(* Schneider Machine Expert - Basic project A7 Temporizador TOF, file version 2.7.0.0 *)
(* ProjectInformations: Name=Novo projeto *)

HARDWARE
  Cpu 0: TM221M16R/G
  EthernetConfiguration: NetworkName=M221, IpAllocationMode=FixedAddress, IpAddress=0.0.0.0, SubnetMask=0.0.0.0
  SerialLineConfiguration: Baud=Baud19200, Parity=ParityEven, DataBits=DataBits8, StopBits=StopBits1, PhysicalMedium=PhysicalMediumRs485, TransmissionMode=TransmissionModeModbusRtu, SlaveId=1, Addressing=SlaveAddressing
  MastTask: UsePeriodScanMode=false, PeriodScan=100
  FastTask: Period=255
  CpuBehavior: StartingMode=StartAsPreviousState, AutoSaveRamOnEeprom=true, WatchdogPeriod=250

SYMBOLS  (address, symbol, comment, settings)
  %TM0        [Type=TOF, Preset=10, Base=OneSecond, IsRetentive=true]

POU Novo POU
  (* SectionNumber=1 *)

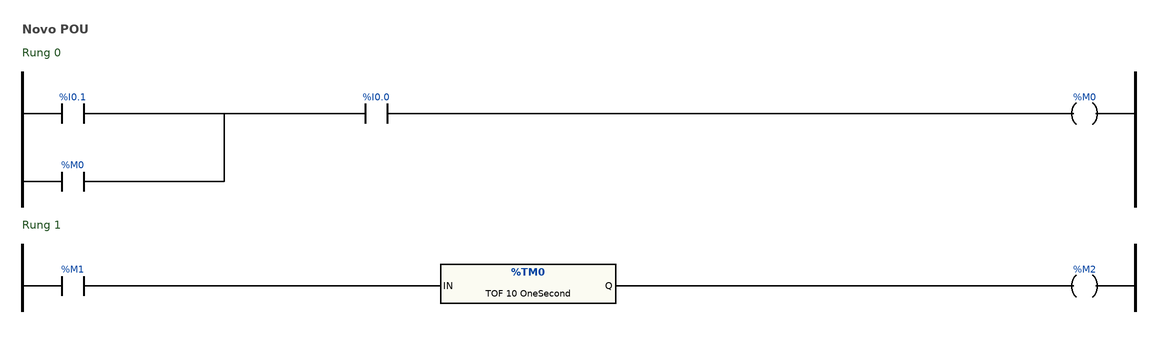

// Rung 0
  LD %I0.1
  OR %M0
  AND %I0.0
  ST %M0
  // as ST:
  //   %M0 := (%I0.1 OR %M0) AND %I0.0;

// Rung 1
  BLK %TM0
  LD %M1
  IN
  OUT_BLK
  LD Q
  ST %M2
  END_BLK
  // as ST:
  //   %TM0(IN := %M1);
  //   %M2 := %TM0.Q;
